FUNCTION F_ComputeDoubleSize : UDINT
VAR_INPUT
    {attribute 'analysis' := '-33' }
    fValue : LREAL;
END_VAR


F_ComputeDoubleSize := GCL_PB.cDoubleSize;

END_FUNCTION

(* stored: Version 1.1.0.1
   POU F_ComputeDoubleSize: Id {c376c301-c279-4a20-9def-68581bb27b67}, SpecialFunc None *)
